(* CoDeSys 2.3 export: RESETPUMPSALARM.EXP *)

(* POU resetPumpsAlarm, ST *)
FUNCTION resetPumpsAlarm : BOOL
(*
	Сброс всех аварий насосов
*)
VAR_INPUT
	IN : BOOL;
END_VAR
VAR
	i : USINT;
END_VAR
IF IN THEN
	FOR i := 1 TO MAX_K14_PUMPS_NUM DO
		K14PumpFaulty[i] := FALSE;
	END_FOR;

	FOR i := 1 TO MAX_K15_PUMPS_NUM DO
		K15PumpFaulty[i] := FALSE;
	END_FOR;

	FOR i := 1 TO MAX_K16_PUMPS_NUM DO
		K16PumpFaulty[i] := FALSE;
	END_FOR;
END_IF;
END_FUNCTION
